FUNCTION_BLOCK FB_ALARM EXTENDS FB_TcAlarm
VAR_INPUT
	eventEntry : TcEventEntry;
	bEvt : BOOL;
	bConfirm : BOOL;
	nUserEventID : UDINT;
	nUserSourceID : UDINT;
	sMessage : STRING;
	sSourceMessage : STRING;
END_VAR
VAR_IN_OUT
	arrAlarms : ARRAY[*] OF TYP_ALARMS;
END_VAR
VAR_OUTPUT
END_VAR
VAR
	bInit : BOOL := TRUE;
	bMem : BOOL;
	fbMsg : FB_TcMessage;
	fbSourceInformation : FB_TcSourceInfo;
END_VAR

//INITIALISING THE ALARM WHEN THE RAISING OF THE ALARM IS REQUESTED
IF bEvt AND NOT bMem (*AND SUPER^.eConfirmationState <> TcEventConfirmationState.WaitForConfirmation*) THEN
	IF bInit THEN
		fbSourceInformation.Clear();
		fbSourceInformation.sName := sSourceMessage;
		fbSourceInformation.nId := nUserSourceID;
		eventEntry.nEventId := nUserEventID;
		SUPER^.CreateEx(eventEntry, TRUE, ipSourceInfo := fbSourceInformation);
		SUPER^.ipArguments.Clear().AddString(sMessage);
		bInit := FALSE;
	END_IF
END_IF

//AFTER INITIALISING, RAISE THE ALARM
IF NOT bInit THEN
	SUPER^.Raise(0);
	bInit := TRUE;
END_IF

//CLEARING THE ALARM
IF bMem AND NOT bEvt THEN
	SUPER^.Clear(0, FALSE);	
END_IF

//CONFIRMING THE ALARM
IF bConfirm THEN
	SUPER^.Confirm(0);
END_IF

bMem := bEvt;

END_FUNCTION_BLOCK

(* stored: Version 1.1.0.1, ProductVersion 3.1.4024.12
   POU FB_ALARM: Id {ab473ddc-b744-4d35-8468-395ce076faea}, SpecialFunc None *)
